# EPICS substitutions: vacuumSimApp/Db/pump.substitutions
# pump substitutions file

file db/turbopump.db {
    pattern { P, V1, V2, G1, G2 }
        { P, V1, V2, G1, G2 }
}
